PROGRAM P_EventLogger_TCSAlarms

//CREATES AND HANDLES ALARMS BASED ON THE WIN WIND ALARM STRUCTURE THAT EXISTS ALREADY
VAR
	fbAlarm:ARRAY[1..222] OF FB_TcAlarm;
	fbSourceInfo : FB_TcSourceInfo;
	binit: BOOL;
	i:UINT; 
	index2:UINT;
END_VAR

initAlarms();
IF bInit THEN
	FOR index2:=1 TO 222 DO
		RaiseAlarms();
		
		ClearAlarms();
	END_FOR
END_IF

ACTION ClearAlarms:
// IF WIN WIND ALARM IS CLEARED, COMMAND THE INSTANCE OF THE CREATE TC3 ALARM TO CLEAR ALSO
IF NOT arrAlarms[index2].b THEN
	 fbAlarm[index2].Clear(0, TRUE);
END_IF
END_ACTION

ACTION initAlarms:
//Initialise alarms based on the brake program defined in the arrAlarms array of ST_ALARMSTRUCTURE
IF NOT binit THEN
	FOR i:=1 TO 222 DO
		CASE arrAlarms[i].eBrakeProgram OF
			B1:
				fbSourceInfo.Clear();
				fbSourceInfo.sName := arrAlarms[i].sName;
				fbAlarm[i].CreateEx(TC_Events.AlarmSystem.B1, FALSE, fbSourceInfo);
			B2:
				fbSourceInfo.Clear();
				fbSourceInfo.sName := arrAlarms[i].sName;
				fbAlarm[i].CreateEx(TC_Events.AlarmSystem.B2, FALSE, fbSourceInfo);
			B3:
				fbSourceInfo.Clear();
				fbSourceInfo.sName := arrAlarms[i].sName;
				fbAlarm[i].CreateEx(TC_Events.AlarmSystem.B3, FALSE, fbSourceInfo);
			B4:
				fbSourceInfo.Clear();
				fbSourceInfo.sName := arrAlarms[i].sName;
				fbAlarm[i].CreateEx(TC_Events.AlarmSystem.B4, FALSE, fbSourceInfo);
			B5:
				fbSourceInfo.Clear();
				fbSourceInfo.sName := arrAlarms[i].sName;
				fbAlarm[i].CreateEx(TC_Events.AlarmSystem.B5, FALSE, fbSourceInfo);
			B6:
				fbSourceInfo.Clear();
				fbSourceInfo.sName := arrAlarms[i].sName;
				fbAlarm[i].CreateEx(TC_Events.AlarmSystem.B6, FALSE, fbSourceInfo);
			B7:
				fbSourceInfo.Clear();
				fbSourceInfo.sName := arrAlarms[i].sName;
				fbAlarm[i].CreateEx(TC_Events.AlarmSystem.B7, FALSE, fbSourceInfo);
			B8:
				fbSourceInfo.Clear();
				fbSourceInfo.sName := arrAlarms[i].sName;
				fbAlarm[i].CreateEx(TC_Events.AlarmSystem.B8, FALSE, fbSourceInfo);
			B9:
				fbSourceInfo.Clear();
				fbSourceInfo.sName := arrAlarms[i].sName;
				fbAlarm[i].CreateEx(TC_Events.AlarmSystem.B9, FALSE, fbSourceInfo);
			B10:
				fbSourceInfo.Clear();
				fbSourceInfo.sName := arrAlarms[i].sName;
				fbAlarm[i].CreateEx(TC_Events.AlarmSystem.B10, FALSE, fbSourceInfo);
			B11:
				fbSourceInfo.Clear();
				fbSourceInfo.sName := arrAlarms[i].sName;
				fbAlarm[i].CreateEx(TC_Events.AlarmSystem.B11, FALSE, fbSourceInfo);
			B12:
				fbSourceInfo.Clear();
				fbSourceInfo.sName := arrAlarms[i].sName;
				fbAlarm[i].CreateEx(TC_Events.AlarmSystem.B12, FALSE, fbSourceInfo);
			B13:
				fbSourceInfo.Clear();
				fbSourceInfo.sName := arrAlarms[i].sName;
				fbAlarm[i].CreateEx(TC_Events.AlarmSystem.B13, FALSE, fbSourceInfo);
			B14:
				fbSourceInfo.Clear();
				fbSourceInfo.sName := arrAlarms[i].sName;
				fbAlarm[i].CreateEx(TC_Events.AlarmSystem.B14, FALSE, fbSourceInfo);
			B15:
				fbSourceInfo.Clear();
				fbSourceInfo.sName := arrAlarms[i].sName;
				fbAlarm[i].CreateEx(TC_Events.AlarmSystem.B15, FALSE, fbSourceInfo);
			B16:
				fbSourceInfo.Clear();
				fbSourceInfo.sName := arrAlarms[i].sName;
				fbAlarm[i].CreateEx(TC_Events.AlarmSystem.B16, FALSE, fbSourceInfo);
			B17:
				fbSourceInfo.Clear();
				fbSourceInfo.sName := arrAlarms[i].sName;
				fbAlarm[i].CreateEx(TC_Events.AlarmSystem.B17, FALSE, fbSourceInfo);
			B18:
				fbSourceInfo.Clear();
				fbSourceInfo.sName := arrAlarms[i].sName;
				fbAlarm[i].CreateEx(TC_Events.AlarmSystem.B18, FALSE, fbSourceInfo);
			B20:
				fbSourceInfo.Clear();
				fbSourceInfo.sName := arrAlarms[i].sName;
				fbAlarm[i].CreateEx(TC_Events.AlarmSystem.B20, FALSE, fbSourceInfo);
			B25:
				fbSourceInfo.Clear();
				fbSourceInfo.sName := arrAlarms[i].sName;
				fbAlarm[i].CreateEx(TC_Events.AlarmSystem.B25, FALSE, fbSourceInfo);
			B30:
				fbSourceInfo.Clear();
				fbSourceInfo.sName := arrAlarms[i].sName;
				fbAlarm[i].CreateEx(TC_Events.AlarmSystem.B30, FALSE, fbSourceInfo);
			B40:
				fbSourceInfo.Clear();
				fbSourceInfo.sName := arrAlarms[i].sName;
				fbAlarm[i].CreateEx(TC_Events.AlarmSystem.B40, FALSE, fbSourceInfo);
			B99:
				fbSourceInfo.Clear();
				fbSourceInfo.sName := arrAlarms[i].sName;
				fbAlarm[i].CreateEx(TC_Events.AlarmSystem.B99, FALSE, fbSourceInfo);
			B100:
				fbSourceInfo.Clear();
				fbSourceInfo.sName := arrAlarms[i].sName;
				fbAlarm[i].CreateEx(TC_Events.AlarmSystem.B100, FALSE, fbSourceInfo);
			
		END_CASE
	END_FOR
	
 IF i>=222 THEN
	 bInit:=1;
 END_IF
END_IF
END_ACTION

ACTION RaiseAlarms:
// COMMAND ALARMS BASED ON THE .B OF THE WIN WIND ALARM STUCTURE
    //bRaiseAlarm[1] := FALSE;
	IF arrAlarms[index2].b THEN
   		fbAlarm[index2].ipArguments.Clear().AddString(arrAlarms[index2].Comment);
    	fbAlarm[index2].Raise(0);
	END_IF
END_ACTION

END_PROGRAM

(* stored: Version 1.1.0.1, ProductVersion 3.1.4024.11
   POU P_EventLogger_TCSAlarms: Id {ad298a10-e02d-4585-bb77-f5a974f8c8da}, SpecialFunc None
   Action ClearAlarms: Id {e0313fea-919f-4672-90ed-89ca6a19030d}
   Action initAlarms: Id {2d07e112-512a-4111-8f7b-521d51bd7454}
   Action RaiseAlarms: Id {74ed3deb-ec15-4c2b-9834-aa170c346b41} *)
